// TIA Portal project "function block1" (V16)

(* hardware
DEVICE "S7-1200 station_1"  S7-1200 Station
   slot 0: "Rack_0"  S7-1200 Rack  Rack  V1.0
   slot 1: "PLC_1"  CPU 1214C DC/DC/DC  6ES7 214-1AG40-0XB0  V4.4
   slot 2: "AI 4x13BIT/AQ 2x14BIT_1"  6ES7 234-4HE32-0XB0  V2.1
   slot 101: "CP 1243-7 LTE"  CP 1243-7 LTE  6GK7 243-7KX30-0XE0  V3.2
      slot 0: "Telecontrol server"  Partner
      slot 0: "Inter-station communication"  Partner
   slot 102: "RF120C_1"  RF120C  6GT2 002-0LA00  V1.0
   slot 103: "CM 1243-5"  CM 1243-5  6GK7 243-5DX30-0XE0  V1.3
*)

// ===== PLC "PLC_1"  CPU 1214C DC/DC/DC =====

VAR_GLOBAL   // PLC tag table "Default tag table"
   "switch" AT %M0.0 : Bool;
   "out" AT %M0.1 : Bool;
   "estop" AT %M0.2 : Bool;
   "esnotification" AT %M0.3 : Bool;
   "esalarm" AT %M0.4 : Bool;
   "alarmreset" AT %M0.5 : Bool;
   "alarmsilent" AT %M0.6 : Bool;
   "val1" AT %MW2 : Int;
   "val3" AT %MW4 : Int;
   "switch2" AT %M0.7 : Bool;
   "reset" AT %M1.0 : Bool;
END_VAR

DATA_BLOCK "scl_DB"   // DB1
{ S7_Optimized_Access := 'TRUE' }
VERSION : 0.1
// stored: InstanceOfName scl
"scl"
BEGIN
END_DATA_BLOCK

FUNCTION_BLOCK "scl"   // FB1, SCL
{ S7_Optimized_Access := 'TRUE' }
VERSION : 0.1
   VAR
      almset : Bool;
      i : Int;
      loopset : Bool;
      loopset2 : Bool;
   END_VAR
   VAR_TEMP
      val2 : Int;
   END_VAR
BEGIN
   IF "switch" AND NOT #loopset THEN
       FOR #i := 0 TO 99 DO
           "val1" := "val1" + 3;
       END_FOR;
       #loopset := 1;
   END_IF;
   IF "switch2" AND NOT #loopset2 THEN
       WHILE "val3" < 6000 DO
           "val3" := "val3" + 1;// Statement section WHILE

       END_WHILE;
       #loopset2 := 1;
   END_IF;
   IF "reset" THEN
       #loopset := 0;
       #loopset2 := 0;
   END_IF;
END_FUNCTION_BLOCK

ORGANIZATION_BLOCK "Main"   // OB1, LAD, ProgramCycle
TITLE = "Main Program Sweep (Cycle)"
{ S7_Optimized_Access := 'TRUE' }
VERSION : 0.1
   VAR_INPUT
      Initial_Call : Bool;   // Initial call of this OB
      Remanence : Bool;   // =True, if remanent data are available
   END_VAR
BEGIN

REGION Network 1
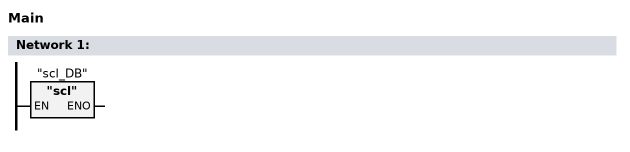
   RUNG wire#powerrail
      "scl_DB"()
   END_RUNG
   // the same network as SCL:
   "scl_DB"();   // "scl"
END_REGION
END_ORGANIZATION_BLOCK